// TIA Portal V17 export
// export: Created 2024-08-29T18:23:51.1234094Z, ExportSetting WithDefaults, DisplayName Totally Integrated Automation Portal, DisplayVersion V17 Update 7, DisplayName TIA Portal Openness, DisplayVersion V17 Update 7, DisplayName TIA Portal Version Control Interface, DisplayVersion V17, DisplayName SINAMICS Startdrive Advanced, DisplayVersion V17 SP2, DisplayName SINAMICS Startdrive G110M, G120, G120C, G120D, G120P, G115D, DisplayVersion V17 SP2, DisplayName SINAMICS Startdrive G130, G150, S120, S150, SINAMICS MV, S210, DisplayVersion V17 SP2, DisplayName STEP 7 Professional, DisplayVersion V17 Update 7, DisplayName STEP 7 Safety, DisplayVersion V17 Update 6, DisplayName WinCC Advanced / Unified PC, DisplayVersion V17 Update 7
TYPE "udt_EKS_KEY"
// stored: IsFailsafeCompliant false
   STRUCT
      ID1 : DWord;   // Key unique ID [bytes 1-4]
      ID2 : DWord;   // Key unique ID [bytes 5-8]
      EMPLOYEE_ID : DWord;   // Employee ID number [hex format]
      LEVEL : Int;   // Key level stored inside key
      COMMENTS : WString[10];   // Comments of the key
      _res_1 : Int;
   END_STRUCT;
END_TYPE
